(* IEC 61131-3 sources: crb-codesys/generation/scripts/repoeval/重型运输系统/can/PRG, 14 files *)

(* ---- CanRx.st ---- *)
PROGRAM CanRx
VAR
	count		:UINT;
END_VAR

count := count + 1;
IF count > 1000 THEN
	count := 1;
END_IF

C01_Rx();
C02_Rx();
C03_Rx();
C04_Rx();
C05_Rx();
C06_Rx();

(* ---- CanRx_C01_Rx_method.st ---- *)
METHOD C01_Rx
VAR_INPUT
END_VAR
VAR
	frame	 	    :Can_baseframe;
	I				:UINT;
	fId				:UINT;
	pos				:WORD;
	spd				:WORD;
END_VAR

IF gCan.C1RxMsg.RxCounter <>  gCan.C1RxCounter THEN    //接收到新的数据
	FOR I := 1 TO gCan.C1RxMsg.NoOfRxMessages DO
		frame := CAN_Read_Data_SWMC(1,I);
		fId := frame.id;
		CASE fId OF
			16#600:
				pos := BYTE_TO_WORD(frame.data[ 1 ]) OR SHL(BYTE_TO_WORD(frame.data[ 2 ]),8);
				gDev.sky[4].sensor.position := pos * 0.1;
				pos := BYTE_TO_WORD(frame.data[ 3 ]) OR SHL(BYTE_TO_WORD(frame.data[ 4 ]),8);
				gDev.sky[5].sensor.position := pos * 0.1;
				pos := BYTE_TO_WORD(frame.data[ 5 ]) OR SHL(BYTE_TO_WORD(frame.data[ 6 ]),8);
				gDev.sky[6].sensor.position := pos * 0.1;
				pos := BYTE_TO_WORD(frame.data[ 7 ]) OR SHL(BYTE_TO_WORD(frame.data[ 8 ]),8);
				gDev.sky[3].sensor.position := pos * 0.1;
			16#601:
				spd := BYTE_TO_WORD(frame.data[ 1 ]) OR SHL(BYTE_TO_WORD(frame.data[ 2 ]),8);
				gDev.sky[4].sensor.speed := INT_TO_REAL(WORD_TO_INT(spd));
				spd := BYTE_TO_WORD(frame.data[ 3 ]) OR SHL(BYTE_TO_WORD(frame.data[ 4 ]),8);
				gDev.sky[5].sensor.speed := INT_TO_REAL(WORD_TO_INT(spd));
				spd := BYTE_TO_WORD(frame.data[ 5 ]) OR SHL(BYTE_TO_WORD(frame.data[ 6 ]),8);
				gDev.sky[6].sensor.speed := INT_TO_REAL(WORD_TO_INT(spd));
				spd := BYTE_TO_WORD(frame.data[ 7 ]) OR SHL(BYTE_TO_WORD(frame.data[ 8 ]),8);
				gDev.sky[3].sensor.speed := INT_TO_REAL(WORD_TO_INT(spd));
		END_CASE

	END_FOR
	gCan.C1RxCounter := gCan.C1RxMsg.RxCounter;
END_IF

(* ---- CanRx_C01_Tx_method.st ---- *)
METHOD C01_Tx
VAR_INPUT
END_VAR
VAR
	swmcIdSwtich		:UINT;
	sendData			:ARRAY[1..8] OF BYTE;
END_VAR

swmcIdSwtich := count MOD 2;
CASE swmcIdSwtich OF
	0:
		sendData[1] := WORD_TO_BYTE(gController.sky[3].extendPercent);
		sendData[2] := WORD_TO_BYTE(SHR(gController.sky[3].extendPercent,8));
		sendData[3] := WORD_TO_BYTE(gController.sky[3].retractPercent);
		sendData[4] := WORD_TO_BYTE(SHR(gController.sky[3].retractPercent,8));
		sendData[5] := WORD_TO_BYTE(gController.sky[4].extendPercent);
		sendData[6] := WORD_TO_BYTE(SHR(gController.sky[4].extendPercent,8));
		sendData[7] := WORD_TO_BYTE(gController.sky[4].retractPercent);
		sendData[8] := WORD_TO_BYTE(SHR(gController.sky[4].retractPercent,8));
		CAN_Send_Data_SWMC(1, 16#500,senddata);   //发送ID 0x460到C6

	1:
		sendData[1] := WORD_TO_BYTE(gController.sky[5].extendPercent);
		sendData[2] := WORD_TO_BYTE(SHR(gController.sky[5].extendPercent,8));
		sendData[3] := WORD_TO_BYTE(gController.sky[5].retractPercent);
		sendData[4] := WORD_TO_BYTE(SHR(gController.sky[5].retractPercent,8));
		sendData[5] := WORD_TO_BYTE(gController.sky[6].extendPercent);
		sendData[6] := WORD_TO_BYTE(SHR(gController.sky[6].extendPercent,8));
		sendData[7] := WORD_TO_BYTE(gController.sky[6].retractPercent);
		sendData[8] := WORD_TO_BYTE(SHR(gController.sky[6].retractPercent,8));
		CAN_Send_Data_SWMC(1, 16#501,senddata);   //发送ID 0x460到C6

END_CASE

(* ---- CanRx_C02_Rx_method.st ---- *)
METHOD C02_Rx
VAR_INPUT
END_VAR
VAR
	frame	 	    :Can_baseframe;
	I				:UINT;
	fId				:UINT;
	pos				:WORD;
	spd				:WORD;
END_VAR

IF gCan.C2RxMsg.RxCounter <>  gCan.C2RxCounter THEN    //接收到新的数据
	FOR I := 1 TO gCan.C2RxMsg.NoOfRxMessages DO
		frame := CAN_Read_Data_SWMC(2,I);
		fId := frame.id;
		CASE fId OF
			16#610:
				pos := BYTE_TO_WORD(frame.data[ 1 ]) OR SHL(BYTE_TO_WORD(frame.data[ 2 ]),8);
				gDev.sky[0].sensor.position := pos * 0.1;
				pos := BYTE_TO_WORD(frame.data[ 3 ]) OR SHL(BYTE_TO_WORD(frame.data[ 4 ]),8);
				gDev.sky[1].sensor.position := pos * 0.1;
				pos := BYTE_TO_WORD(frame.data[ 5 ]) OR SHL(BYTE_TO_WORD(frame.data[ 6 ]),8);
				gDev.sky[2].sensor.position := pos * 0.1;

			16#611:
				spd := BYTE_TO_WORD(frame.data[ 1 ]) OR SHL(BYTE_TO_WORD(frame.data[ 2 ]),8);
				gDev.sky[0].sensor.speed := INT_TO_REAL(WORD_TO_INT(spd));
				spd := BYTE_TO_WORD(frame.data[ 3 ]) OR SHL(BYTE_TO_WORD(frame.data[ 4 ]),8);
				gDev.sky[1].sensor.speed := INT_TO_REAL(WORD_TO_INT(spd));
				spd := BYTE_TO_WORD(frame.data[ 5 ]) OR SHL(BYTE_TO_WORD(frame.data[ 6 ]),8);
				gDev.sky[2].sensor.speed := INT_TO_REAL(WORD_TO_INT(spd));
		END_CASE
	END_FOR
	gCan.C2RxCounter := gCan.C2RxMsg.RxCounter;
END_IF

(* ---- CanRx_C02_Tx_method.st ---- *)
METHOD C02_Tx
VAR_INPUT
END_VAR
VAR
	swmcIdSwtich		:UINT;
	sendData			:ARRAY[1..8] OF BYTE;
END_VAR

swmcIdSwtich := count MOD 2;
CASE swmcIdSwtich OF
	0:
		sendData[1] := WORD_TO_BYTE(gController.sky[0].extendPercent);
		sendData[2] := WORD_TO_BYTE(SHR(gController.sky[0].extendPercent,8));
		sendData[3] := WORD_TO_BYTE(gController.sky[0].retractPercent);
		sendData[4] := WORD_TO_BYTE(SHR(gController.sky[0].retractPercent,8));
		sendData[5] := WORD_TO_BYTE(gController.sky[1].extendPercent);
		sendData[6] := WORD_TO_BYTE(SHR(gController.sky[1].extendPercent,8));
		sendData[7] := WORD_TO_BYTE(gController.sky[1].retractPercent);
		sendData[8] := WORD_TO_BYTE(SHR(gController.sky[1].retractPercent,8));
		CAN_Send_Data_SWMC(2, 16#510,senddata);   //发送ID 0x460到C6

	1:
		sendData[1] := WORD_TO_BYTE(gController.sky[2].extendPercent);
		sendData[2] := WORD_TO_BYTE(SHR(gController.sky[2].extendPercent,8));
		sendData[3] := WORD_TO_BYTE(gController.sky[2].retractPercent);
		sendData[4] := WORD_TO_BYTE(SHR(gController.sky[2].retractPercent,8));
		CAN_Send_Data_SWMC(2, 16#511,senddata);   //发送ID 0x460到C6

END_CASE

(* ---- CanRx_C03_Rx_method.st ---- *)
METHOD C03_Rx
VAR_INPUT
END_VAR
VAR
	frame	 	    :Can_baseframe;
	I				:UINT;
	fId				:UINT;
	pos				:WORD;
	spd				:WORD;
	cur				:WORD;	//current
END_VAR

IF gCan.C3RxMsg.RxCounter <>  gCan.C3RxCounter THEN    //接收到新的数据
	FOR I := 1 TO gCan.C3RxMsg.NoOfRxMessages DO
		frame := CAN_Read_Data_SWMC(3,I);
		fId := frame.id;
		CASE fId OF
			16#620:
				pos := BYTE_TO_WORD(frame.data[ 1 ]) OR SHL(BYTE_TO_WORD(frame.data[ 2 ]),8);
				gDev.grd[5].sensor.position := pos * 0.1;
				pos := BYTE_TO_WORD(frame.data[ 3 ]) OR SHL(BYTE_TO_WORD(frame.data[ 4 ]),8);
				gDev.grd[6].sensor.position := pos * 0.1;
				pos := BYTE_TO_WORD(frame.data[ 5 ]) OR SHL(BYTE_TO_WORD(frame.data[ 6 ]),8);
				gDev.grd[3].sensor.position := pos * 0.1;
				pos := BYTE_TO_WORD(frame.data[ 7 ]) OR SHL(BYTE_TO_WORD(frame.data[ 8 ]),8);
				gDev.grd[4].sensor.position := pos * 0.1;
			16#621:
				spd := BYTE_TO_WORD(frame.data[ 1 ]) OR SHL(BYTE_TO_WORD(frame.data[ 2 ]),8);
				gDev.grd[5].sensor.speed := INT_TO_REAL(WORD_TO_INT(spd));
				spd := BYTE_TO_WORD(frame.data[ 3 ]) OR SHL(BYTE_TO_WORD(frame.data[ 4 ]),8);
				gDev.grd[6].sensor.speed := INT_TO_REAL(WORD_TO_INT(spd));
				spd := BYTE_TO_WORD(frame.data[ 5 ]) OR SHL(BYTE_TO_WORD(frame.data[ 6 ]),8);
				gDev.grd[3].sensor.speed := INT_TO_REAL(WORD_TO_INT(spd));
				spd := BYTE_TO_WORD(frame.data[ 7 ]) OR SHL(BYTE_TO_WORD(frame.data[ 8 ]),8);
				gDev.grd[4].sensor.speed := INT_TO_REAL(WORD_TO_INT(spd));
			16#622:
				cur := BYTE_TO_WORD(frame.data[ 1 ]) OR SHL(BYTE_TO_WORD(frame.data[ 2 ]),8);
				gDev.grd[3].current[1] := cur;
				cur := BYTE_TO_WORD(frame.data[ 3 ]) OR SHL(BYTE_TO_WORD(frame.data[ 4 ]),8);
				gDev.grd[3].current[2] := cur;
				cur := BYTE_TO_WORD(frame.data[ 5 ]) OR SHL(BYTE_TO_WORD(frame.data[ 6 ]),8);
				gDev.grd[4].current[1] := cur;
				cur := BYTE_TO_WORD(frame.data[ 7 ]) OR SHL(BYTE_TO_WORD(frame.data[ 8 ]),8);
				gDev.grd[4].current[2] := cur;
			16#623:
				cur := BYTE_TO_WORD(frame.data[ 1 ]) OR SHL(BYTE_TO_WORD(frame.data[ 2 ]),8);
				gDev.grd[5].current[1] := cur;
				cur := BYTE_TO_WORD(frame.data[ 3 ]) OR SHL(BYTE_TO_WORD(frame.data[ 4 ]),8);
				gDev.grd[5].current[2] := cur;
				cur := BYTE_TO_WORD(frame.data[ 5 ]) OR SHL(BYTE_TO_WORD(frame.data[ 6 ]),8);
				gDev.grd[6].current[1] := cur;
				cur := BYTE_TO_WORD(frame.data[ 7 ]) OR SHL(BYTE_TO_WORD(frame.data[ 8 ]),8);
				gDev.grd[6].current[2] := cur;

		END_CASE
	END_FOR
	gCan.C3RxCounter := gCan.C3RxMsg.RxCounter;
END_IF

(* ---- CanRx_C03_Tx_method.st ---- *)
METHOD C03_Tx
VAR_INPUT
END_VAR
VAR
	swmcIdSwtich		:UINT;
	sendData			:ARRAY[1..8] OF BYTE;
END_VAR

swmcIdSwtich := count MOD 2;
CASE swmcIdSwtich OF
	0:
		sendData[1] := WORD_TO_BYTE(gController.grd[3].extendPercent);
		sendData[2] := WORD_TO_BYTE(SHR(gController.grd[3].extendPercent,8));
		sendData[3] := WORD_TO_BYTE(gController.grd[3].retractPercent);
		sendData[4] := WORD_TO_BYTE(SHR(gController.grd[3].retractPercent,8));
		sendData[5] := WORD_TO_BYTE(gController.grd[4].extendPercent);
		sendData[6] := WORD_TO_BYTE(SHR(gController.grd[4].extendPercent,8));
		sendData[7] := WORD_TO_BYTE(gController.grd[4].retractPercent);
		sendData[8] := WORD_TO_BYTE(SHR(gController.grd[4].retractPercent,8));
		CAN_Send_Data_SWMC(3, 16#520,senddata);   //发送ID 0x460到C6

	1:
		sendData[1] := WORD_TO_BYTE(gController.grd[5].extendPercent);
		sendData[2] := WORD_TO_BYTE(SHR(gController.grd[5].extendPercent,8));
		sendData[3] := WORD_TO_BYTE(gController.grd[5].retractPercent);
		sendData[4] := WORD_TO_BYTE(SHR(gController.grd[5].retractPercent,8));
		sendData[5] := WORD_TO_BYTE(gController.grd[6].extendPercent);
		sendData[6] := WORD_TO_BYTE(SHR(gController.grd[6].extendPercent,8));
		sendData[7] := WORD_TO_BYTE(gController.grd[6].retractPercent);
		sendData[8] := WORD_TO_BYTE(SHR(gController.grd[6].retractPercent,8));
		CAN_Send_Data_SWMC(3, 16#521,senddata);   //发送ID 0x460到C6

END_CASE

(* ---- CanRx_C04_Rx_method.st ---- *)
METHOD C04_Rx
VAR_INPUT
END_VAR
VAR
	frame	 	    :Can_baseframe;
	I				:UINT;
	fId				:UINT;
	pos				:WORD;
	spd				:WORD;

END_VAR

IF gCan.C4RxMsg.RxCounter <>  gCan.C4RxCounter THEN    //接收到新的数据
	FOR I := 1 TO gCan.C4RxMsg.NoOfRxMessages DO
		frame := CAN_Read_Data_SWMC(4,I);
		fId := frame.id;
		CASE fId OF
			16#630:
				pos := BYTE_TO_WORD(frame.data[ 1 ]) OR SHL(BYTE_TO_WORD(frame.data[ 2 ]),8);
				gDev.grd[1].sensor.position := pos * 0.1;
				pos := BYTE_TO_WORD(frame.data[ 3 ]) OR SHL(BYTE_TO_WORD(frame.data[ 4 ]),8);
				gDev.grd[2].sensor.position := pos * 0.1;

			16#631:
				spd := BYTE_TO_WORD(frame.data[ 1 ]) OR SHL(BYTE_TO_WORD(frame.data[ 2 ]),8);
				gDev.grd[1].sensor.speed := INT_TO_REAL(WORD_TO_INT(spd));
				spd := BYTE_TO_WORD(frame.data[ 3 ]) OR SHL(BYTE_TO_WORD(frame.data[ 4 ]),8);
				gDev.grd[2].sensor.speed := INT_TO_REAL(WORD_TO_INT(spd));
		END_CASE
	END_FOR
	gCan.C4RxCounter := gCan.C4RxMsg.RxCounter;
END_IF

(* ---- CanRx_C04_Tx_method.st ---- *)
METHOD C04_Tx
VAR_INPUT
END_VAR
VAR
	swmcIdSwtich		:UINT;
	sendData			:ARRAY[1..8] OF BYTE;
END_VAR

swmcIdSwtich := count MOD 2;
CASE swmcIdSwtich OF
	0:
		sendData[1] := WORD_TO_BYTE(gController.grd[1].extendPercent);
		sendData[2] := WORD_TO_BYTE(SHR(gController.grd[1].extendPercent,8));
		sendData[3] := WORD_TO_BYTE(gController.grd[1].retractPercent);
		sendData[4] := WORD_TO_BYTE(SHR(gController.grd[1].retractPercent,8));
		sendData[5] := WORD_TO_BYTE(gController.grd[2].extendPercent);
		sendData[6] := WORD_TO_BYTE(SHR(gController.grd[2].extendPercent,8));
		sendData[7] := WORD_TO_BYTE(gController.grd[2].retractPercent);
		sendData[8] := WORD_TO_BYTE(SHR(gController.grd[2].retractPercent,8));
		CAN_Send_Data_SWMC(4, 16#530,senddata);   //发送ID 0x460到C6

END_CASE

(* ---- CanRx_C05_Rx_method.st ---- *)
METHOD C05_Rx
VAR_INPUT
END_VAR
VAR
	frame	 	    :Can_baseframe;
	I				:UINT;
	fId				:UINT;
	pos				:WORD;	//位置
	spd				:WORD;	//速度
END_VAR

IF gCan.C5RxMsg.RxCounter <>  gCan.C5RxCounter THEN    //接收到新的数据
	FOR I := 1 TO gCan.C5RxMsg.NoOfRxMessages DO
		frame := CAN_Read_Data_SWMC(5,I);
		fId := frame.id;
		CASE fId OF
			16#640:
				pos := BYTE_TO_WORD(frame.data[ 1 ]) OR SHL(BYTE_TO_WORD(frame.data[ 2 ]),8);
				gDev.sky[7].sensor.position := pos * 0.1;
				pos := BYTE_TO_WORD(frame.data[ 3 ]) OR SHL(BYTE_TO_WORD(frame.data[ 4 ]),8);
				gDev.sky[8].sensor.position := pos * 0.1;
				pos := BYTE_TO_WORD(frame.data[ 5 ]) OR SHL(BYTE_TO_WORD(frame.data[ 6 ]),8);
				gDev.sky[9].sensor.position := pos * 0.1;
				pos := BYTE_TO_WORD(frame.data[ 7 ]) OR SHL(BYTE_TO_WORD(frame.data[ 8 ]),8);
				gDev.sky[10].sensor.position := pos * 0.1;
			16#641:
				spd := BYTE_TO_WORD(frame.data[ 1 ]) OR SHL(BYTE_TO_WORD(frame.data[ 2 ]),8);
				gDev.sky[7].sensor.speed := INT_TO_REAL(WORD_TO_INT(spd));
				spd := BYTE_TO_WORD(frame.data[ 3 ]) OR SHL(BYTE_TO_WORD(frame.data[ 4 ]),8);
				gDev.sky[8].sensor.speed := INT_TO_REAL(WORD_TO_INT(spd));
				spd := BYTE_TO_WORD(frame.data[ 5 ]) OR SHL(BYTE_TO_WORD(frame.data[ 6 ]),8);
				gDev.sky[9].sensor.speed := INT_TO_REAL(WORD_TO_INT(spd));
				spd := BYTE_TO_WORD(frame.data[ 7 ]) OR SHL(BYTE_TO_WORD(frame.data[ 8 ]),8);
				gDev.sky[10].sensor.speed := INT_TO_REAL(WORD_TO_INT(spd));
		END_CASE

	END_FOR
	gCan.C5RxCounter := gCan.C5RxMsg.RxCounter;
END_IF

(* ---- CanRx_C05_Tx_method.st ---- *)
METHOD C05_Tx
VAR_INPUT
END_VAR
VAR
	swmcIdSwtich		:UINT;
	sendData			:ARRAY[1..8] OF BYTE;
END_VAR

swmcIdSwtich := count MOD 2;
CASE swmcIdSwtich OF
	0:
		sendData[1] := WORD_TO_BYTE(gController.sky[7].extendPercent);
		sendData[2] := WORD_TO_BYTE(SHR(gController.sky[7].extendPercent,8));
		sendData[3] := WORD_TO_BYTE(gController.sky[7].retractPercent);
		sendData[4] := WORD_TO_BYTE(SHR(gController.sky[7].retractPercent,8));
		sendData[5] := WORD_TO_BYTE(gController.sky[8].extendPercent);
		sendData[6] := WORD_TO_BYTE(SHR(gController.sky[8].extendPercent,8));
		sendData[7] := WORD_TO_BYTE(gController.sky[8].retractPercent);
		sendData[8] := WORD_TO_BYTE(SHR(gController.sky[8].retractPercent,8));
		CAN_Send_Data_SWMC(5, 16#540,senddata);   //发送ID 0x460到C6
	1:
		sendData[1] := WORD_TO_BYTE(gController.sky[9].extendPercent);
		sendData[2] := WORD_TO_BYTE(SHR(gController.sky[9].extendPercent,8));
		sendData[3] := WORD_TO_BYTE(gController.sky[9].retractPercent);
		sendData[4] := WORD_TO_BYTE(SHR(gController.sky[9].retractPercent,8));
		sendData[5] := WORD_TO_BYTE(gController.sky[10].extendPercent);
		sendData[6] := WORD_TO_BYTE(SHR(gController.sky[10].extendPercent,8));
		sendData[7] := WORD_TO_BYTE(gController.sky[10].retractPercent);
		sendData[8] := WORD_TO_BYTE(SHR(gController.sky[10].retractPercent,8));
		CAN_Send_Data_SWMC(5, 16#541,senddata);   //发送ID 0x460到C6

END_CASE

(* ---- CanRx_C06_Rx_method.st ---- *)
METHOD C06_Rx
VAR_INPUT
END_VAR
VAR
	frame	 	    :Can_baseframe;
	I				:UINT;
	fId				:UINT;
	pos				:WORD;	//位置
	spd				:WORD;	//速度
END_VAR

IF gCan.C6RxMsg.RxCounter <>  gCan.C6RxCounter THEN    //接收到新的数据
	FOR I := 1 TO gCan.C6RxMsg.NoOfRxMessages DO
		frame := CAN_Read_Data_SWMC(6,I);
		fId := frame.id;
		CASE fId OF
			16#650:
				pos := BYTE_TO_WORD(frame.data[ 1 ]) OR SHL(BYTE_TO_WORD(frame.data[ 2 ]),8);
				gDev.grd[7].sensor.position := pos * 0.1;
				pos := BYTE_TO_WORD(frame.data[ 3 ]) OR SHL(BYTE_TO_WORD(frame.data[ 4 ]),8);
				gDev.grd[8].sensor.position := pos * 0.1;
				pos := BYTE_TO_WORD(frame.data[ 5 ]) OR SHL(BYTE_TO_WORD(frame.data[ 6 ]),8);
				gDev.grd[9].sensor.position := pos * 0.1;
				pos := BYTE_TO_WORD(frame.data[ 7 ]) OR SHL(BYTE_TO_WORD(frame.data[ 8 ]),8);
				gDev.grd[10].sensor.position := pos * 0.1;
			16#651:
				spd := BYTE_TO_WORD(frame.data[ 1 ]) OR SHL(BYTE_TO_WORD(frame.data[ 2 ]),8);
				gDev.grd[7].sensor.speed := INT_TO_REAL(WORD_TO_INT(spd));
				spd := BYTE_TO_WORD(frame.data[ 3 ]) OR SHL(BYTE_TO_WORD(frame.data[ 4 ]),8);
				gDev.grd[8].sensor.speed := INT_TO_REAL(WORD_TO_INT(spd));
				spd := BYTE_TO_WORD(frame.data[ 5 ]) OR SHL(BYTE_TO_WORD(frame.data[ 6 ]),8);
				gDev.grd[9].sensor.speed := INT_TO_REAL(WORD_TO_INT(spd));
				spd := BYTE_TO_WORD(frame.data[ 7 ]) OR SHL(BYTE_TO_WORD(frame.data[ 8 ]),8);
				gDev.grd[10].sensor.speed := INT_TO_REAL(WORD_TO_INT(spd));
		END_CASE
	END_FOR
	gCan.C6RxCounter := gCan.C6RxMsg.RxCounter;
END_IF

(* ---- CanRx_C06_Tx_method.st ---- *)
METHOD C06_Tx
VAR_INPUT
END_VAR
VAR
	swmcIdSwtich		:UINT;
	sendData			:ARRAY[1..8] OF BYTE;
END_VAR

swmcIdSwtich := count MOD 2;
CASE swmcIdSwtich OF
	0:
		sendData[1] := WORD_TO_BYTE(gController.grd[7].extendPercent);
		sendData[2] := WORD_TO_BYTE(SHR(gController.grd[7].extendPercent,8));
		sendData[3] := WORD_TO_BYTE(gController.grd[7].retractPercent);
		sendData[4] := WORD_TO_BYTE(SHR(gController.grd[7].retractPercent,8));
		sendData[5] := WORD_TO_BYTE(gController.grd[8].extendPercent);
		sendData[6] := WORD_TO_BYTE(SHR(gController.grd[8].extendPercent,8));
		sendData[7] := WORD_TO_BYTE(gController.grd[8].retractPercent);
		sendData[8] := WORD_TO_BYTE(SHR(gController.grd[8].retractPercent,8));
		CAN_Send_Data_SWMC(6, 16#550,senddata);   //发送ID 0x460到C6

	1:
		sendData[1] := WORD_TO_BYTE(gController.grd[9].extendPercent);
		sendData[2] := WORD_TO_BYTE(SHR(gController.grd[9].extendPercent,8));
		sendData[3] := WORD_TO_BYTE(gController.grd[9].retractPercent);
		sendData[4] := WORD_TO_BYTE(SHR(gController.grd[9].retractPercent,8));
		sendData[5] := WORD_TO_BYTE(gController.grd[10].extendPercent);
		sendData[6] := WORD_TO_BYTE(SHR(gController.grd[10].extendPercent,8));
		sendData[7] := WORD_TO_BYTE(gController.grd[10].retractPercent);
		sendData[8] := WORD_TO_BYTE(SHR(gController.grd[10].retractPercent,8));
		CAN_Send_Data_SWMC(6, 16#551,senddata);   //发送ID 0x460到C6

END_CASE

(* ---- CanTx.st ---- *)
PROGRAM CanTx
VAR
	count		:UINT;
END_VAR

count := count + 1;
IF count > 1000 THEN
	count := 1;
END_IF

C01_Tx();
C02_Tx();
C03_Tx();
C04_Tx();
C05_Tx();
C06_Tx();
